(* CODESYS project beer inputs.project

Project tree, tasks and I/O mapping:
  Device : CODESYS Control Win V3 x64, 3S - Smart Software Solutions GmbH, version 3.5.11.0
    application Application
      libraries: Standard, * (System); VisuDialogs, * (System); Util, * (System)
      task MainTask (cyclic, interval t#10ms, priority 1) calls Plant, Controller
      program Plant [ST]
      global variables GVL
      program Controller [ST]
      visualisation Visualization
      image pool ImagePool
  text list GlobalTextList
  5ce3da45-db07-42e7-a21c-a00fff4ed8f6|C:\Users\fish\Downloads\voenbilet.png
  5ce3da45-db07-42e7-a21c-a00fff4ed8f6|C:\Users\fish\Downloads\jaguar.png
  5ce3da45-db07-42e7-a21c-a00fff4ed8f6|C:\Users\fish\Downloads\monster.png
  5ce3da45-db07-42e7-a21c-a00fff4ed8f6|C:\Users\fish\Downloads\beer.png
  5ce3da45-db07-42e7-a21c-a00fff4ed8f6|C:\Users\fish\Downloads\greencard.png
  5ce3da45-db07-42e7-a21c-a00fff4ed8f6|C:\Users\fish\Downloads\pistol.png
  5ce3da45-db07-42e7-a21c-a00fff4ed8f6|C:\Users\fish\Downloads\cigaretes after vki .png
  5ce3da45-db07-42e7-a21c-a00fff4ed8f6|C:\Users\fish\Documents\MAX.png
*)

// Device/Application/GVL
VAR_GLOBAL
	// Sensors:
	onfloor0:BOOL;		// Elevator at floor 0
	onfloor1:BOOL;		// Elevator at floor 1
	onfloor2:BOOL;		// Elevator at floor 2
	door0closed:BOOL;	// Doors at floor 0 are closed
	door1closed:BOOL;	// Doors at floor 1 are closed
	door2closed:BOOL;	// Doors at floor 2 are closed
	button0:BOOL;		// Call button at floor 0
	button1:BOOL;		// Call button at floor 1
	button2:BOOL;		// Call button at floor 2
	call0:BOOL;			// Request floor 0 from inside the cabin 
	call1:BOOL;			// Request floor 1 from inside the cabin
	call2:BOOL;			// Request floor 2 from inside the cabin
	
	// Actuators:
	up:BOOL;			// Control the elevator to go up
	down:BOOL;			// Control the elevator to go down
	open0:BOOL;			// Open the doors at floor 0
	open1:BOOL;			// Open the doors at floor 1
	open2:BOOL;			// Open the doors at floor 2
	
	call0_LED : BOOL;
	call1_LED : BOOL;
	call2_LED : BOOL;
	
	button0_LED : BOOL;
	button1_LED : BOOL;
	button2_LED : BOOL;
	
	floor0_LED : BOOL;
	floor1_LED : BOOL;
	floor2_LED : BOOL;
	
	cur : INT;
END_VAR

// Device/Application/Plant
PROGRAM Plant

VAR
	Obj : ARRAY[1..5] OF BOOL := [TRUE];
	Drop_control : BOOL := FALSE;
	Button : ARRAY[1..5] OF BOOL := [FALSE];
	Cancellation : BOOL := FALSE;
	bank_terminal : UDINT := 0;
	cash_terminal : UDINT := 0;
	user: INT;
END_VAR

VAR
	MAX_call : BOOL;
	i : INT;
	Drop_obj : ARRAY[1..5] OF BOOL;
	tratit_bank : BOOL := FALSE;
	kopit_bank : BOOL := FALSE;
	user_bank : UDINT := 0;
	user_change : UDINT := 0;
	tovar : ARRAY[1..5] OF INT := [3, 3, 3, 3, 3];
END_VAR

IF kopit_bank THEN
	user_bank := user_bank + 1;
	kopit_bank := FALSE;
END_IF
IF tratit_bank THEN
	IF user_bank > 0 THEN 
		user_bank := user_bank - 1;
	END_IF
	tratit_bank := FALSE;
END_IF
IF Cancellation THEN
	user_change := user_change + cash_terminal;
	cash_terminal := 0;
END_IF

FOR i := 1 TO 5 DO
	Obj[i] := tovar[i] > 0;
END_FOR;

FOR i := 1 TO 5 DO
	IF Drop_obj[i] THEN
		tovar[i] := MAX(tovar[i] - 1, 0);
		Drop_obj[i] := FALSE;
	END_IF
END_FOR;

IF MAX_call THEN
	FOR i := 1 TO 5 DO
		tovar[i] := 3;
	END_FOR;
END_IF

END_PROGRAM

// Device/Application/Controller
PROGRAM Controller

VAR CONSTANT
	_STOP : INT := 254;
	_ERROR : INT := 255;
END_VAR

VAR
	target : INT;
END_VAR

END_PROGRAM

// Device/Application/Visualization
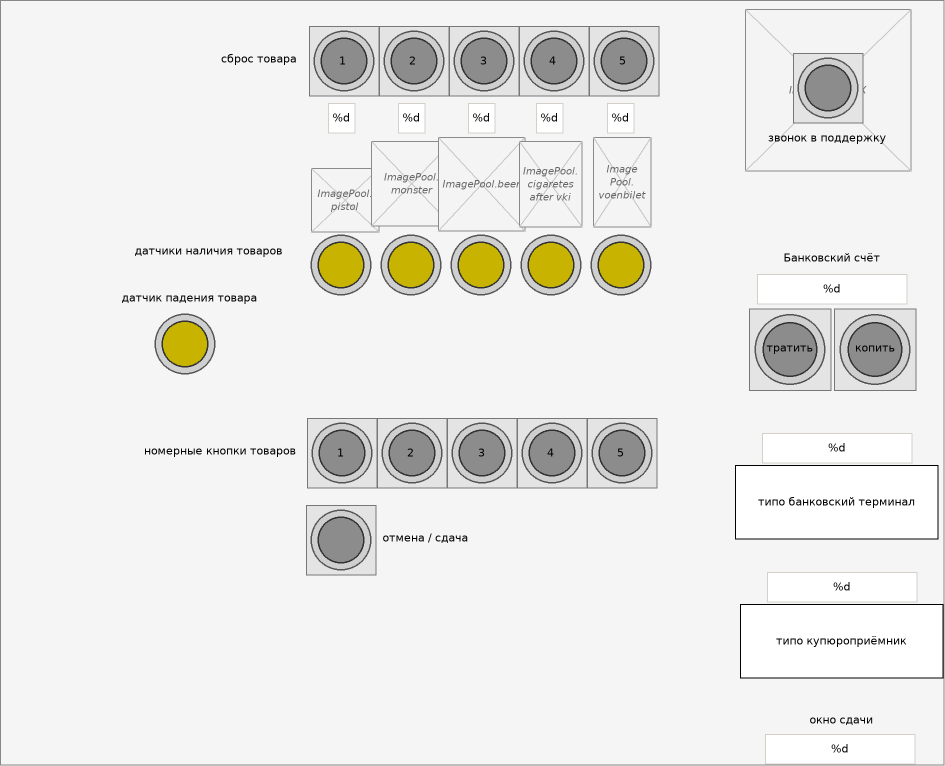
VISUALIZATION Visualization  // 945x766
IN_OUT
	
END_VAR
    Image (745,9 166x162), image: ImagePool.MAX
    Lamp1 (306,230 70x70), variable: Plant.Obj[1], style: Lamp-Lamp1-Yellow
    Lamp1 (376,230 70x70), variable: Plant.Obj[2], style: Lamp-Lamp1-Yellow
    Lamp1 (446,230 70x70), variable: Plant.Obj[3], style: Lamp-Lamp1-Yellow
    Lamp1 (516,230 70x70), variable: Plant.Obj[4], style: Lamp-Lamp1-Yellow
    Lamp1 (586,230 70x70), variable: Plant.Obj[5], style: Lamp-Lamp1-Yellow
    Label (126,224 169x54), "датчики наличия товаров"
    Label (757,243 150x30), "Банковский счёт"
    Textfield (757,274 150x30), "%d", text variable: Plant.user_bank
    PushSwitch (834,308 82x83), tooltip "на порш", variable: Plant.kopit_bank, behaviour: TOGGLE, style: Switch-PushSwitch-Gray
    Label (840,333 70x30), "копить"
    PushSwitch (749,308 82x83), tooltip "платно?", variable: Plant.tratit_bank, behaviour: TOGGLE, style: Switch-PushSwitch-Gray
    Label (755,333 70x30), "тратить"
    Label (839,486 70x30)
    Rectangle (735,465 203x74), "типо банковский терминал"
        OnMouseLeave: execute { Plant.bank_terminal := 0; }
        OnMouseEnter: execute { Plant.bank_terminal := Plant.user_bank; }
    Textfield (762,433 150x30), "%d", text variable: Plant.bank_terminal
    Rectangle (740,604 203x74), "типо купюроприёмник"
        OnMouseClick: execute { Plant.cash_terminal := Plant.cash_terminal + 5; }
    Textfield (767,572 150x30), "%d", text variable: Plant.cash_terminal
    PushSwitch (307,418 70x70), tooltip "платно?", variable: Plant.Button[1], behaviour: TAP, style: Switch-PushSwitch-Gray
    PushSwitch (377,418 70x70), tooltip "платно?", variable: Plant.Button[2], behaviour: TAP, style: Switch-PushSwitch-Gray
    PushSwitch (587,418 70x70), tooltip "платно?", variable: Plant.Button[5], behaviour: TAP, style: Switch-PushSwitch-Gray
    PushSwitch (517,418 70x70), tooltip "платно?", variable: Plant.Button[4], behaviour: TAP, style: Switch-PushSwitch-Gray
    PushSwitch (447,418 70x70), tooltip "платно?", variable: Plant.Button[3], behaviour: TAP, style: Switch-PushSwitch-Gray
    Label (137,424 166x54), "номерные кнопки товаров"
    Label (317,426 47x54), "1"
    Label (387,426 47x54), "2"
    Label (458,426 47x54), "3"
    Label (527,426 47x54), "4"
    Label (597,426 47x54), "5"
    PushSwitch (306,505 70x70), tooltip "платно?", variable: Plant.Cancellation, behaviour: TAP, style: Switch-PushSwitch-Gray
    Label (370,511 111x54), "отмена / сдача"
    Lamp1 (150,309 70x70), variable: Plant.Drop_control, style: Lamp-Lamp1-Yellow
    Label (118,271 143x54), "датчик падения товара"
    Textfield (765,734 150x30), "%d", tooltip "забрать сдачу", text variable: Plant.user_change
        OnMouseClick: execute { Plant.user_change := 0; }
    Label (786,693 111x54), "окно сдачи"
    Image (311,168 68x64), angle 35, image: ImagePool.pistol
    Image (371,141 81x85), angle 2, image: ImagePool.monster
    Image (438,137 87x94), image: ImagePool.beer
    Image (593,137 58x90), image: ImagePool.voenbilet
    Textfield (328,103 27x30), "%d", text variable: Plant.tovar[1]
    Image (519,141 63x86), image: ImagePool.cigaretes after vki
    Textfield (398,103 27x30), "%d", text variable: Plant.tovar[2]
    Textfield (468,103 27x30), "%d", text variable: Plant.tovar[3]
    Textfield (536,103 27x30), "%d", text variable: Plant.tovar[4]
    Textfield (607,103 27x30), "%d", text variable: Plant.tovar[5]
    PushSwitch (309,26 70x70), tooltip "платно?", variable: Plant.Drop_obj[1], behaviour: TAP, style: Switch-PushSwitch-Gray
    PushSwitch (379,26 70x70), tooltip "платно?", variable: Plant.Drop_obj[2], behaviour: TAP, style: Switch-PushSwitch-Gray
    PushSwitch (589,26 70x70), tooltip "платно?", variable: Plant.Drop_obj[5], behaviour: TAP, style: Switch-PushSwitch-Gray
    PushSwitch (519,26 70x70), tooltip "платно?", variable: Plant.Drop_obj[4], behaviour: TAP, style: Switch-PushSwitch-Gray
    PushSwitch (449,26 70x70), tooltip "платно?", variable: Plant.Drop_obj[3], behaviour: TAP, style: Switch-PushSwitch-Gray
    Label (319,34 47x54), "1"
    Label (389,34 47x54), "2"
    Label (460,34 47x54), "3"
    Label (529,34 47x54), "4"
    Label (599,34 47x54), "5"
    Label (176,32 166x54), "сброс товара"
    PushSwitch (793,53 70x70), tooltip "*только в MAX", variable: Plant.MAX_call, behaviour: TAP, style: Switch-PushSwitch-Gray
    Label (744,111 166x54), "звонок в поддержку"
END_VISUALIZATION
